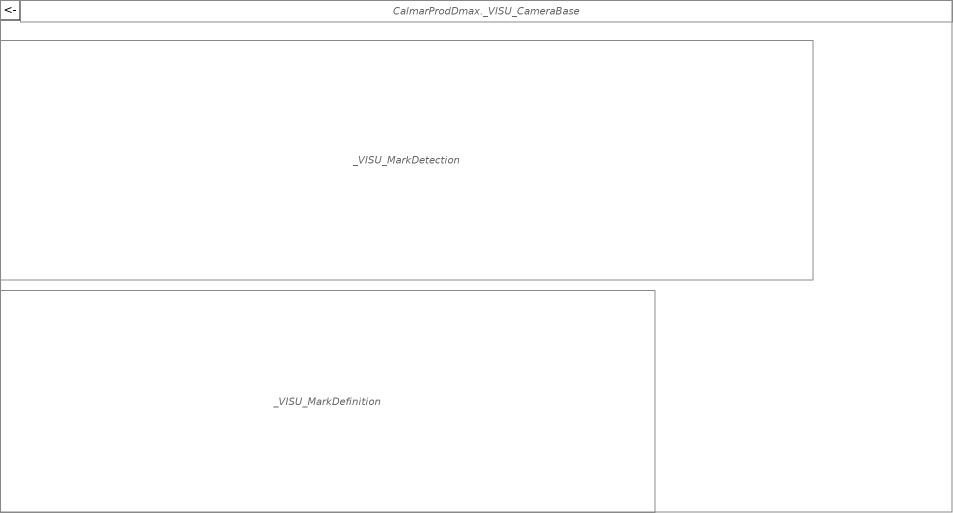
VISUALIZATION _VISU_MarkCamera_WEU  // 953x513
VAR_IN_OUT
  mCam : FB_MarkCamera_WEU;
  mMarkDetect : FB_MarkDetection;
END_VAR
    RoundedRectangle (0,0 20x20), "<-"
        OnMouseClick: change screen: Previous 
    Frame (0,290 655x223)
        shows _VISU_MarkDefinition(mInst := mMarkDetect._pFbMarkDefinition^)
    Frame (20,0 933x22)
        shows CalmarProdDmax._VISU_CameraBase(m_Inst := mCam)
    Frame (0,40 813x240)
        shows _VISU_MarkDetection(mInst := mMarkDetect)
END_VISUALIZATION

(* stored: Version 1.1.0.1, ProductVersion 3.1.4024.11
   Visu _VISU_MarkCamera_WEU: Id {9f70e9c9-8020-455c-86cd-0e0b18206fdf} *)
